Yaskawa INFORM job: X2_24A(90,180).JBI

/JOB
//NAME X2_24A(90,180)
///FOLDERNAME X2
//POS
///NPOS 98,98,98,6,0,0
///TOOL 0
///POSTYPE PULSE
///PULSE
C00000=2000,-92772,-84335,0,66375,0
C00001=-61786,-92772,-84335,-2347,66375,79401
C00002=-97244,21725,-41177,22449,93615,82233
C00003=-95530,462,4396,55956,36816,51794
C00004=-94424,6187,12285,57576,35067,50925
C00005=-93996,8571,15581,58338,34366,50524
C00006=-93996,9261,17575,59445,33898,49925
C00007=-93996,8571,15581,58338,34366,50524
C00008=-93267,12817,19373,58151,33839,50654
C00009=-93996,8571,15581,58338,34366,50524
C00010=-95521,1087,6495,57044,36258,51187
C00011=-96592,2869,6453,65825,56052,48227
C00012=-94772,6998,13020,66731,54034,47573
C00013=-94060,8748,15768,67150,53233,47286
C00014=-94060,9552,18085,67847,52819,46755
C00015=-94060,8748,15768,67150,53233,47286
C00016=-92626,10057,16930,66950,52266,47512
C00017=-94060,8748,15768,67150,53233,47286
C00018=-96573,3490,8496,66397,55638,47762
C00019=-83582,5061,8367,59913,58634,65118
C00020=-81471,7687,13629,60535,56339,64672
C00021=-80635,8836,15839,60828,55424,64478
C00022=-80635,9690,18292,61474,54884,63961
C00023=-80635,8836,15839,60828,55424,64478
C00024=-79828,9033,16014,60679,54915,64642
C00025=-80635,8836,15839,60828,55424,64478
C00026=-83597,5664,10366,60398,58167,64691
C00027=-83314,10150,12730,59594,89568,59936
C00028=-81399,9267,14976,59682,87415,59552
C00029=-81014,9626,17081,59725,86592,59179
C00030=-81014,10332,19089,59751,86136,58834
C00031=-81014,9626,17081,59725,86592,59179
C00032=-80226,8223,15841,59775,86122,59334
C00033=-81014,9626,17081,59725,86592,59179
C00034=-83301,10774,14815,59578,89053,59559
C00035=-98806,-6617,-7331,59053,101140,58606
C00036=-97102,-16285,-8510,58460,97807,57230
C00037=-95610,-19203,-5710,58231,95144,56240
C00038=-95610,-18645,-4180,58161,94786,55981
C00039=-96019,-16166,-2121,59216,96428,56839
C00040=-95765,-17656,-3227,59244,96227,56851
C00041=-96019,-16166,-2121,59216,96428,56839
C00042=-98806,-6617,-7331,59053,101140,58606
C00043=-83650,45812,10891,63097,77396,50083
C00044=-82040,46827,21520,63951,73569,47805
C00045=-81304,48087,22594,63748,73022,47936
C00046=-82382,46154,21930,64152,73438,47516
C00047=-81304,48083,24007,63975,72618,47565
C00048=-79820,39299,14734,60932,66880,49784
C00049=-80553,45924,21635,60013,63961,50168
C00050=-80159,45513,21016,56886,58795,52013
C00051=-79446,45138,20749,53508,54059,53881
C00052=-80802,51037,27110,52596,51762,54266
C00053=-80810,51549,27463,50423,49544,55420
C00054=-80796,51959,27984,49530,48507,55881
C00055=-80807,52184,28258,48800,47721,56262
C00056=-80745,52371,28448,47312,46281,57045
C00057=-80076,50770,26686,45255,44934,58131
C00058=-80548,47424,22156,44596,45760,58565
C00059=-81458,42877,14387,43611,47989,59314
C00060=-91002,51772,6505,49273,82170,67204
C00061=-101987,13091,-892,55645,108662,64355
C00062=-110253,6769,-1127,53677,111646,61313
C00063=-109069,2020,-4496,53719,110740,61430
C00064=-109385,7501,2227,53217,110114,60832
C00065=-109069,2458,-2118,53294,109982,60937
C00066=-100675,7100,1874,54374,105065,62741
C00067=-99850,8509,2883,54486,104646,62955
C00068=-98291,5259,89,55265,98561,65120
C00069=-92725,-3222,-7154,54399,80249,71381
C00070=-87115,-4435,-8234,50482,66809,76551
C00071=-92539,-2221,-10635,51205,72117,76021
C00072=-96871,14274,1468,54076,82371,72764
C00073=-94701,9031,3178,59274,52046,46005
C00074=-93342,13775,10378,60199,50156,45313
C00075=-92447,15859,11447,59599,49816,45723
C00076=-93434,13866,11409,60652,49914,44989
C00077=-92447,16412,13741,60428,49230,45145
C00078=-92744,16958,14199,60523,49416,45077
C00079=-95754,24729,21609,57662,43562,46984
C00080=-96395,24314,20911,42110,30641,55727
C00081=-96416,20010,16135,41713,31228,55971
C00082=-96977,14076,7690,40003,33138,56882
C00083=-85021,42815,2038,36976,67324,74168
C00084=-87037,99,-8557,56339,77378,69862
C00085=-84861,88,-5624,56340,75042,69589
C00086=-84770,-1894,-7034,56357,74898,69547
C00087=-86315,-1244,-5605,56691,75514,69027
C00088=-84770,-1696,-5978,56472,74585,69332
C00089=-84707,-1124,-5491,56466,74544,69342
C00090=-83566,14086,7749,56369,73673,69438
C00091=-81991,21704,14907,53912,65153,72184
C00092=-78809,22027,15079,45737,51427,78665
C00093=-78646,18844,10981,44406,51004,79638
C00094=-80451,15982,5388,44195,53341,79866
C00095=-97244,21725,-41177,22449,93615,82233
C00096=-75987,-111338,-91135,3036,61075,74073
C00097=2000,-92772,-84335,0,66375,0
BC00000=244954,666204,804590
BC00001=244954,672262,286248
BC00002=244954,696126,53
BC00003=305530,775472,205864
BC00004=305530,775472,205864
BC00005=305530,775472,205864
BC00006=305530,775472,205864
BC00007=305530,775472,205864
BC00008=305530,775472,205864
BC00009=305530,775472,205864
BC00010=305530,775472,205864
BC00011=306859,760141,205932
BC00012=306859,760141,205932
BC00013=306859,760141,205932
BC00014=306859,760141,205932
BC00015=306859,760141,205932
BC00016=306859,760141,205932
BC00017=306859,760141,205932
BC00018=306859,760141,205932
BC00019=266237,742564,232226
BC00020=266237,742564,232226
BC00021=266237,742564,232226
BC00022=266237,742564,232226
BC00023=266237,742564,232226
BC00024=266237,742564,232226
BC00025=266237,742564,232226
BC00026=266237,742564,232226
BC00027=250497,756280,248827
BC00028=250497,756280,248827
BC00029=250497,756280,248827
BC00030=250497,756280,248827
BC00031=250497,756280,248827
BC00032=250497,756280,248827
BC00033=250497,756280,248827
BC00034=250497,756280,248827
BC00035=250497,756280,248827
BC00036=250497,756280,248827
BC00037=250497,756280,248827
BC00038=250497,756280,248827
BC00039=250497,756280,248827
BC00040=250497,756280,248827
BC00041=250497,756280,248827
BC00042=250497,756280,248827
BC00043=252145,743870,53
BC00044=252145,743870,53
BC00045=252145,743870,53
BC00046=252145,743870,53
BC00047=252145,743870,53
BC00048=252145,743870,53
BC00049=252145,743870,53
BC00050=252145,743870,53
BC00051=252145,743870,53
BC00052=252145,743870,53
BC00053=252145,743870,53
BC00054=252145,743870,53
BC00055=252145,743870,53
BC00056=252145,743870,53
BC00057=252145,743870,53
BC00058=252145,743870,53
BC00059=252145,743870,53
BC00060=254165,705505,53
BC00061=278436,722364,176042
BC00062=278436,722364,176042
BC00063=278436,722364,176042
BC00064=278436,722364,176042
BC00065=278436,722364,176042
BC00066=278436,722364,176042
BC00067=278436,722364,176042
BC00068=278436,722364,176042
BC00069=278436,722364,176040
BC00070=278436,722364,176042
BC00071=278436,722364,176042
BC00072=278436,722364,176042
BC00073=300797,766702,142606
BC00074=300797,766702,142606
BC00075=300797,766702,142600
BC00076=300797,766702,142600
BC00077=300797,766702,142600
BC00078=300797,766702,142602
BC00079=300797,766702,142606
BC00080=300797,766702,142606
BC00081=300797,766702,142606
BC00082=300797,766702,142606
BC00083=248658,714848,53
BC00084=269872,740220,162373
BC00085=269872,740220,162373
BC00086=269872,740220,162373
BC00087=269872,740220,162373
BC00088=269872,740220,162373
BC00089=269872,740220,162373
BC00090=269872,740220,162373
BC00091=269872,740220,162373
BC00092=269872,740220,162373
BC00093=269872,740220,162373
BC00094=269872,740220,162373
BC00095=244954,696126,53
BC00096=244954,672262,286248
BC00097=244954,666204,804590
EC00000=798156,1112951
EC00001=798156,1112951
EC00002=798156,1112951
EC00003=798156,1112951
EC00004=798156,1112951
EC00005=798156,1112951
EC00006=798156,1112951
EC00007=798156,1112951
EC00008=798156,1112951
EC00009=798156,1112951
EC00010=798156,1112951
EC00011=798156,1112951
EC00012=798156,1112951
EC00013=798156,1112951
EC00014=798156,1112951
EC00015=798156,1112951
EC00016=798156,1112951
EC00017=798156,1112951
EC00018=798156,1112951
EC00019=798156,1112951
EC00020=798156,1112951
EC00021=798156,1112951
EC00022=798156,1112951
EC00023=798156,1112951
EC00024=798156,1112951
EC00025=798156,1112951
EC00026=798156,1112951
EC00027=798156,1112951
EC00028=798156,1112951
EC00029=798156,1112951
EC00030=798156,1112951
EC00031=798156,1112951
EC00032=798156,1112951
EC00033=798156,1112951
EC00034=798156,1112951
EC00035=798156,1112951
EC00036=798156,1112951
EC00037=798156,1112951
EC00038=798156,1112951
EC00039=798156,1112951
EC00040=798156,1112951
EC00041=798156,1112951
EC00042=798156,1112951
EC00043=798156,1112951
EC00044=798156,1112951
EC00045=798156,1112951
EC00046=798156,1112951
EC00047=798156,1112951
EC00048=798156,1112951
EC00049=798156,1112951
EC00050=798156,1112951
EC00051=798156,1112951
EC00052=798156,1112951
EC00053=798156,1112951
EC00054=798156,1112951
EC00055=798156,1112951
EC00056=798156,1112951
EC00057=798156,1112951
EC00058=798156,1112951
EC00059=798156,1112951
EC00060=798156,1112951
EC00061=798156,1112951
EC00062=798156,1112951
EC00063=798156,1112951
EC00064=798156,1112951
EC00065=798156,1112951
EC00066=798156,1112951
EC00067=798156,1112951
EC00068=798156,1112951
EC00069=798155,1112950
EC00070=798156,1112951
EC00071=798156,1112951
EC00072=798156,1112951
EC00073=798156,1112951
EC00074=798156,1112951
EC00075=798154,1112949
EC00076=798154,1112949
EC00077=798154,1112949
EC00078=798155,1112949
EC00079=798156,1112951
EC00080=798156,1112951
EC00081=798156,1112951
EC00082=798156,1112951
EC00083=798156,1112951
EC00084=798156,1112951
EC00085=798156,1112951
EC00086=798156,1112951
EC00087=798156,1112951
EC00088=798156,1112951
EC00089=798156,1112951
EC00090=798156,1112951
EC00091=798156,1112951
EC00092=798156,1112951
EC00093=798156,1112951
EC00094=798156,1112951
EC00095=798156,1112951
EC00096=798156,1112951
EC00097=798156,1112951
///POSTYPE BASE
///RECTAN
///RCONF 0,0,0,0,0,0,0,0,0,0,0,0,0,0,0,0,0,0,0,0,0,0,0,0
P00006=0.222,-3.123,-1.508,0.0000,0.0000,0.0000
P00021=-0.225,-6.128,-0.405,0.0000,0.0000,0.0000
P00022=0.222,-3.123,-1.508,0.0000,0.0000,0.0000
P00023=0.143,-0.036,0.682,0.0000,0.0000,0.0000
P00024=0.145,-0.552,1.326,0.0000,0.0000,0.0000
P00025=-2.003,0.006,0.728,0.0000,0.0000,0.0000
//INST
///DATE 2024/04/06 13:59
///ATTR SC,RW
///GROUP1 RB1,BS1
///GROUP2 ST1
NOP
'X2_24A(90,180)
MOVJ C00000 BC00000 VJ=100.00  +MOVJ EC00000 VJ=100.00
MOVJ C00001 BC00001 VJ=100.00  +MOVJ EC00001 VJ=100.00
MOVJ C00002 BC00002 VJ=100.00  +MOVJ EC00002 VJ=100.00
'Path S3533
SFTOF3D
MOVJ C00003 BC00003 VJ=100.00  +MOVJ EC00003 VJ=100.00
MOVL C00004 BC00004 V=800.0  +MOVJ EC00004 VJ=100.00
SMOVL C00005 BC00005 V=166.7  +MOVJ EC00005
SREFP 3 C00006 BC00006  +REFP EC00006
CALL JOB:SEARCH-R1-S13D
SET P021 P006
SFTON3D P021
SMOVL C00007 BC00007 V=166.7  +MOVJ EC00007
SREFP 3 C00008 BC00008  +REFP EC00008
CALL JOB:SEARCH-R1-S13D
SET P021 P006
SFTON3D P021
SMOVL C00009 BC00009 V=166.7  +MOVJ EC00009
MOVL C00010 BC00010 V=1000.0  +MOVJ EC00010 VJ=100.00
'EndPath S3533
'Path S3534
SFTOF3D
MOVJ C00011 BC00011 VJ=100.00  +MOVJ EC00011 VJ=100.00
MOVL C00012 BC00012 V=800.0  +MOVJ EC00012 VJ=100.00
SMOVL C00013 BC00013 V=166.7  +MOVJ EC00013
SREFP 3 C00014 BC00014  +REFP EC00014
CALL JOB:SEARCH-R1-S13D
SET P022 P006
SFTON3D P022
SMOVL C00015 BC00015 V=166.7  +MOVJ EC00015
SREFP 3 C00016 BC00016  +REFP EC00016
CALL JOB:SEARCH-R1-S13D
SET P022 P006
SFTON3D P022
SMOVL C00017 BC00017 V=166.7  +MOVJ EC00017
MOVL C00018 BC00018 V=1000.0  +MOVJ EC00018 VJ=100.00
'EndPath S3534
'Path S3535
SFTOF3D
MOVJ C00019 BC00019 VJ=100.00  +MOVJ EC00019 VJ=100.00
MOVL C00020 BC00020 V=800.0  +MOVJ EC00020 VJ=100.00
SMOVL C00021 BC00021 V=166.7  +MOVJ EC00021
SREFP 3 C00022 BC00022  +REFP EC00022
CALL JOB:SEARCH-R1-S13D
SET P023 P006
SFTON3D P023
SMOVL C00023 BC00023 V=166.7  +MOVJ EC00023
SREFP 3 C00024 BC00024  +REFP EC00024
CALL JOB:SEARCH-R1-S13D
SET P023 P006
SFTON3D P023
SMOVL C00025 BC00025 V=166.7  +MOVJ EC00025
MOVL C00026 BC00026 V=1000.0  +MOVJ EC00026 VJ=100.00
'EndPath S3535
'Path S3536
SFTOF3D
MOVJ C00027 BC00027 VJ=100.00  +MOVJ EC00027 VJ=100.00
MOVL C00028 BC00028 V=800.0  +MOVJ EC00028 VJ=100.00
SMOVL C00029 BC00029 V=166.7  +MOVJ EC00029
SREFP 3 C00030 BC00030  +REFP EC00030
CALL JOB:SEARCH-R1-S13D
SET P024 P006
SFTON3D P024
SMOVL C00031 BC00031 V=166.7  +MOVJ EC00031
SREFP 3 C00032 BC00032  +REFP EC00032
CALL JOB:SEARCH-R1-S13D
SET P024 P006
SFTON3D P024
SMOVL C00033 BC00033 V=166.7  +MOVJ EC00033
MOVL C00034 BC00034 V=1000.0  +MOVJ EC00034 VJ=100.00
'EndPath S3536
'Path W3537
SFTOF3D
MOVJ C00035 BC00035 VJ=100.00  +MOVJ EC00035 VJ=100.00
MOVL C00036 BC00036 V=800.0  +MOVJ EC00036 VJ=100.00
SMOVL C00037 BC00037 V=166.7  +MOVJ EC00037
SREFP 3 C00038 BC00038  +REFP EC00038
CALL JOB:SEARCH-R1-S13D
SET P025 P006
SFTON3D P025
SMOVL C00039 BC00039 V=166.7  +MOVJ EC00039
SREFP 3 C00040 BC00040  +REFP EC00040
CALL JOB:SEARCH-R1-S13D
SET P025 P006
SFTON3D P025
SMOVL C00041 BC00041 V=166.7  +MOVJ EC00041
MOVL C00042 BC00042 V=1000.0  +MOVJ EC00042 VJ=100.00
SFTOF3D
SFTON3D P022
MOVJ C00043 BC00043 VJ=100.00  +MOVJ EC00043 VJ=100.00
SMOVL C00044 BC00044 V=800.0  +MOVJ EC00044
SREFP 1 C00045 BC00045  +REFP EC00045
SREFP 2 C00046 BC00046  +REFP EC00046
SMOVL C00047 BC00047 V=150.0 PL=0  +MOVJ EC00047
MACRO1 MJ#(0) ARGF21
ARCON
SWVON WEV#(100)
SMOVC C00048 BC00048 V=9.2  +MOVJ EC00048
SMOVC C00049 BC00049 V=9.2  +MOVJ EC00049
SMOVC C00050 BC00050 V=9.2  +MOVJ EC00050
SMOVC C00051 BC00051 V=9.2  +MOVJ EC00051
SMOVC C00052 BC00052 V=9.2  +MOVJ EC00052
ARCON
SWVON WEV#(100)
SMOVC C00053 BC00053 V=9.2  +MOVJ EC00053
SMOVC C00054 BC00054 V=9.2  +MOVJ EC00054
SMOVC C00055 BC00055 V=9.2  +MOVJ EC00055
SMOVC C00056 BC00056 V=9.2  +MOVJ EC00056
SMOVC C00057 BC00057 V=9.2  +MOVJ EC00057
ARCOF
SWVOF
SMOVL C00058 BC00058 V=800.0  +MOVJ EC00058
SMOVL C00059 BC00059 V=1000.0  +MOVJ EC00059
SFTOF3D
'EndPath W3537
MOVJ C00060 BC00060 VJ=100.00  +MOVJ EC00060 VJ=100.00
'Path W3538
SFTOF3D
SFTON3D P025
MOVJ C00061 BC00061 VJ=100.00  +MOVJ EC00061 VJ=100.00
SMOVL C00062 BC00062 V=800.0  +MOVJ EC00062
SREFP 1 C00063 BC00063  +REFP EC00063
SREFP 2 C00064 BC00064  +REFP EC00064
SMOVL C00065 BC00065 V=150.0 PL=0  +MOVJ EC00065
ARCON
SWVON WEV#(100)
SMOVL C00066 BC00066 V=9.2  +MOVJ EC00066
SMOVC C00067 BC00067 V=9.2  +MOVJ EC00067
SFTON3D P024
SMOVC C00068 BC00068 V=9.2  +MOVJ EC00068
SMOVC C00069 BC00069 V=9.2  +MOVJ EC00069
SMOVC C00070 BC00070 V=9.2  +MOVJ EC00070
ARCOF
SWVOF
SMOVL C00071 BC00071 V=800.0  +MOVJ EC00071
SMOVL C00072 BC00072 V=1000.0  +MOVJ EC00072
SFTOF3D
'EndPath W3538
'Path W3539
SFTOF3D
SFTON3D P021
MOVJ C00073 BC00073 VJ=100.00  +MOVJ EC00073 VJ=100.00
SMOVL C00074 BC00074 V=800.0  +MOVJ EC00074
SREFP 1 C00075 BC00075  +REFP EC00075
SREFP 2 C00076 BC00076  +REFP EC00076
SMOVL C00077 BC00077 V=150.0 PL=0  +MOVJ EC00077
ARCON
SWVON WEV#(100)
SMOVC C00078 BC00078 V=9.2  +MOVJ EC00078
SMOVC C00079 BC00079 V=9.2  +MOVJ EC00079
SMOVC C00080 BC00080 V=9.2  +MOVJ EC00080
ARCOF
SWVOF
SMOVL C00081 BC00081 V=800.0  +MOVJ EC00081
SMOVL C00082 BC00082 V=1000.0  +MOVJ EC00082
SFTOF3D
'EndPath W3539
MOVJ C00083 BC00083 VJ=100.00  +MOVJ EC00083 VJ=100.00
'Path W3540
SFTOF3D
SFTON3D P023
MOVJ C00084 BC00084 VJ=100.00  +MOVJ EC00084 VJ=100.00
SMOVL C00085 BC00085 V=800.0  +MOVJ EC00085
SREFP 1 C00086 BC00086  +REFP EC00086
SREFP 2 C00087 BC00087  +REFP EC00087
SMOVL C00088 BC00088 V=166.7 PL=0  +MOVJ EC00088
ARCON
SWVON WEV#(100)
SMOVC C00089 BC00089 V=9.2  +MOVJ EC00089
SMOVC C00090 BC00090 V=9.2  +MOVJ EC00090
SMOVC C00091 BC00091 V=9.2  +MOVJ EC00091
SMOVC C00092 BC00092 V=9.2  +MOVJ EC00092
ARCOF
SWVOF
SMOVL C00093 BC00093 V=800.0  +MOVJ EC00093
SMOVL C00094 BC00094 V=1000.0  +MOVJ EC00094
SFTOF3D
'EndPath W3540
MOVJ C00095 BC00095 VJ=100.00  +MOVJ EC00095 VJ=100.00
MOVJ C00096 BC00096 VJ=100.00  +MOVJ EC00096 VJ=100.00
MOVJ C00097 BC00097 VJ=100.00  +MOVJ EC00097 VJ=100.00
END
